// TIA Portal V20 export
DATA_BLOCK "Simulation"   // DB134
TITLE = Simulation
// Simulation data
// stored: MemoryReserve 100
   VAR
      data : "LAF_typeSimulation";
      hmiSimulationAxis { S7_SetPoint := 'True'} : Array[0..10] of LReal;
   END_VAR
BEGIN
END_DATA_BLOCK
